INTERFACE I_Application

PROPERTY fbLog : REFERENCE TO FB_LogFifo
GET
END_GET
SET
END_SET
END_PROPERTY

PROPERTY fbRx : REFERENCE TO FB_FrameFifo
GET
END_GET
SET
END_SET
END_PROPERTY

PROPERTY fbTx : REFERENCE TO FB_FrameFifo
GET
END_GET
SET
END_SET
END_PROPERTY

PROPERTY isUpdated : bool
GET
END_GET
END_PROPERTY

METHOD Receive
END_METHOD

METHOD Send
END_METHOD

END_INTERFACE

(* stored: Version 1.1.0.1, ProductVersion 3.1.4024.12
   Itf I_Application: Id {7c07e586-e693-443d-86aa-8d247af267c7}
   Property fbLog: Id {5f4aa1b6-d35d-4b8e-a375-e4a45eea418c}
   Get Get: Id {d75206dc-060f-48e5-8894-e508cc6e3b04}
   Set Set: Id {1454964c-0632-4943-92e0-6bf9ce0e9b3c}
   Property fbRx: Id {0b06efa2-7795-4f7f-8a2f-c4fb05fab6cf}
   Get Get: Id {64661e22-a942-42a3-85da-7178e2c2b709}
   Set Set: Id {7567ceda-2f5d-4068-8c32-e3c41fbe82b5}
   Property fbTx: Id {1b5165b1-bac7-47bf-9e0e-9ab393cb8e85}
   Get Get: Id {f00841e2-7680-491b-8d8e-3923ac910717}
   Set Set: Id {e7a02768-8093-4d54-abff-bf5355596e80}
   Property isUpdated: Id {ec43008f-4899-45d3-8609-d0a5f65169ac}
   Get Get: Id {625a3793-0b55-4768-86a2-ac43e79f2345}
   Method Receive: Id {34b5a84c-a02a-4728-964b-2416a738d0a8}
   Method Send: Id {5cc328a4-8b67-4ac8-9aa5-ac1d87afda76} *)
